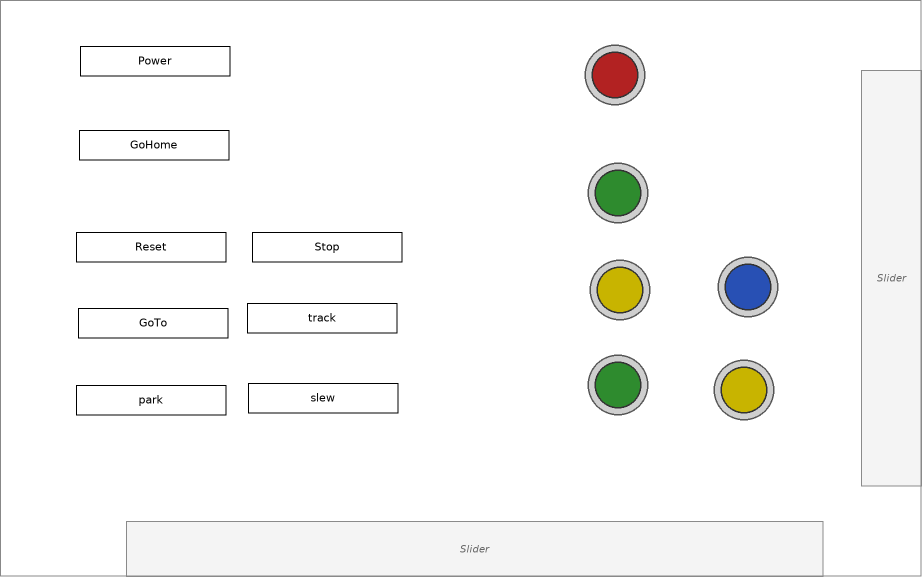
VISUALIZATION Visualization  // 922x577
    RoundedRectangle (80,46 150x30), "Power", colour toggle: TelescopeControl.power
        toggle TelescopeControl.power
    Rectangle (79,130 150x30), "GoHome", colour toggle: TelescopeControl.gohome
        toggle TelescopeControl.gohome
    Lamp1 (580,40 70x70), tooltip "Error", variable: TelescopeControl.error, style: Lamp-Lamp1-Red
    Lamp1 (583,158 70x70), tooltip "ready", variable: TelescopeControl.ready, style: Lamp-Lamp1-Green
    Rectangle (76,232 150x30), "Reset", colour toggle: TelescopeControl.reset
        toggle TelescopeControl.reset
    RoundedRectangle (78,308 150x30), "GoTo", colour toggle: TelescopeControl.goto
        toggle TelescopeControl.goto
    Lamp1 (585,255 70x70), tooltip "sliding", variable: TelescopeControl.sliding, style: Lamp-Lamp1-Yellow
    RoundedRectangle (76,385 150x30), "park", colour toggle: TelescopeControl.park
        toggle TelescopeControl.park
    Lamp1 (583,350 70x70), tooltip "stopped", variable: TelescopeControl.Safetypped, style: Lamp-Lamp1-Green
    Slider (126,521 697x56), variable: TelescopeControl.rightascension, scale 0..360
    Slider (861,70 61x416), variable: TelescopeControl.declination, scale -90..90
    Lamp1 (713,252 70x70), tooltip "tracking", variable: TelescopeControl.tracking, style: Lamp-Lamp1-Blue
    RoundedRectangle (247,303 150x30), "track", colour toggle: TelescopeControl.track
        toggle TelescopeControl.track
    RoundedRectangle (248,383 150x30), "slew", colour toggle: TelescopeControl.slew
        toggle TelescopeControl.slew
    Lamp1 (709,355 70x70), tooltip "busy", variable: TelescopeControl.busy, style: Lamp-Lamp1-Yellow
    RoundedRectangle (252,232 150x30), "Stop", colour toggle: TelescopeControl.Safetyp
        toggle TelescopeControl.stop
END_VISUALIZATION

(* stored: Version 1.1.0.1, ProductVersion 3.1.4026.8
   Visu Visualization: Id {8f6f0973-3e4b-4d5a-8717-02ae98399bab} *)
